FUNCTION_BLOCK THRESHOLD (* openCV threshold *)
  (* Version 1.0, AN, SWDC RTSoft *)
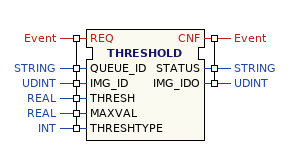
  EVENT_INPUT
    REQ WITH QUEUE_ID, IMG_ID, THRESH, MAXVAL, THRESHTYPE;
  END_EVENT
  EVENT_OUTPUT
    CNF WITH STATUS, IMG_IDO;
  END_EVENT
  VAR_INPUT
    QUEUE_ID : STRING;
    IMG_ID : UDINT;
    THRESH : REAL;
    MAXVAL : REAL;
    THRESHTYPE : INT; (* Threshold type. 0: Binary Inv, 1: Binary, 2: ToZero Inv, 3: ToZero, 4: Trunc *)
  END_VAR
  VAR_OUTPUT
    STATUS : STRING;
    IMG_IDO : UDINT;
  END_VAR
  ALGORITHM REQ IN ST:

  END_ALGORITHM
END_FUNCTION_BLOCK
